// TIA Portal project "032_500_Analog_Values_V14" (V14)

(* hardware
DEVICE "S71500/ET200MP station_1"  S7-1500 station
   slot 0: "Rail_0"  Rack  6ES7 590-1***0-0AA0
   slot 0: "PM 190W 120/230VAC"  PM 190W 120/230VAC  6EP1333-4BA00
   slot 1: "CPU1516F"  CPU 1516F-3 PN/DP  6ES7 516-3FN01-0AB0  V2.1
      slot 3: "CPU display_1"  6ES7591-1BA00-0AA0
   slot 2: "DI 32x24VDC HF_1"  DI 32x24VDC HF  6ES7 521-1BL00-0AB0  V2.1
   slot 3: "DQ 32x24VDC/0.5A HF_1"  DQ 32x24VDC/0.5A HF  6ES7 522-1BL01-0AB0  V1.0
   slot 4: "AI 8xU/I/RTD/TC ST_1"  AI 8xU/I/RTD/TC ST  6ES7 531-7KF00-0AB0  V2.1
   slot 5: "AQ 4xU/I ST_1"  AQ 4xU/I ST  6ES7 532-5HD00-0AB0  V2.1
*)

// ===== PLC "CPU1516F"  CPU 1516F-3 PN/DP =====

VAR_GLOBAL   // PLC tag table "Tag table_sorting station"
   "-A1" AT %I0.0 : Bool;   // return signal emergency stop ok (nc)
   "-K0" AT %I0.1 : Bool;   // main switch „ON“ (no)
   "-S0" AT %I0.2 : Bool;   // mode selector manual(0) / automatic(1)
   "-S1" AT %I0.3 : Bool;   // pushbutton automatic start (no)
   "-S2" AT %I0.4 : Bool;   // pushbutton automatic stop (nc)
   "-B1" AT %I0.5 : Bool;   // sensor cylinder -M4 retracted (no)
   "-B2" AT %I0.6 : Bool;   // sensor cylinder -M4 extended (nc)
   "-B3" AT %I0.7 : Bool;   // sensor motor -M1 actice (pulse signal for positioning) (no)
   "-B4" AT %I1.0 : Bool;   // sensor part at slide (no)
   "-B5" AT %I1.1 : Bool;   // sensor metal part (no)
   "-B6" AT %I1.2 : Bool;   // sensor part in front of cylinder -M4 (no)
   "-B7" AT %I1.3 : Bool;   // sensor part at end of conveyor (no)
   "-S3" AT %I1.4 : Bool;   // pushbutton manual mode conveyor –M1 forwards (no)
   "-S4" AT %I1.5 : Bool;   // pushbutton manual mode conveyor –M1 backwards (no)
   "-S5" AT %I1.6 : Bool;   // pushbutton manual mode cylinder -M4 retract (no)
   "-S6" AT %I1.7 : Bool;   // pushbutton manual mode cylinder -M4 extend (no)
   "-Q1" AT %Q0.0 : Bool;   // conveyor motor -M1 forwards fixed speed
   "-Q2" AT %Q0.1 : Bool;   // conveyor motor -M1 backwards fixed speed
   "-Q3" AT %Q0.2 : Bool;   // conveyor motor -M1 variable speed
   "-M2" AT %Q0.3 : Bool;   // cylinder -M4 retract
   "-M3" AT %Q0.4 : Bool;   // cylinder -M4 extend
   "-P1" AT %Q0.5 : Bool;   // display „main switch on“
   "-P2" AT %Q0.6 : Bool;   // display „manual mode“
   "-P3" AT %Q0.7 : Bool;   // display „automatic mode“
   "-P4" AT %Q1.0 : Bool;   // display „emergency stop activated“
   "-P5" AT %Q1.1 : Bool;   // display „automatic mode started“
   "-P6" AT %Q1.2 : Bool;   // display cylinder -M4 „retracted“
   "-P7" AT %Q1.3 : Bool;   // display cylinder -M4 „extended“
   "-U1" AT %AW64 : Int;   // manipulated value speed in 2 directions +/- 10V / Stellwert Drehzahl des Motors in 2 Richtungen +/-10V entsprechen +/- 50 U/min
   "-B8" AT %EW64 : Int;   // sensor actual value speed 0 …10V / Sensor Istwert Drehzahl des Motors +/-10V entsprechen +/- 50 U/min
END_VAR

DATA_BLOCK "MOTOR_AUTO_DB"   // DB1
{ S7_Optimized_Access := 'TRUE' }
VERSION : 0.1
// stored: InstanceOfName MOTOR_AUTO
"MOTOR_AUTO"
BEGIN
END_DATA_BLOCK

FUNCTION_BLOCK "MOTOR_AUTO"   // FB1, FBD
TITLE = Motor control in automatic mode / Motoransteuerung im Automatikbetrieb
{ S7_Optimized_Access := 'TRUE' }
VERSION : 0.1
// Conveyor motor in automatic mode:
// The bit  Memory_automatic_start_stop is set with the input Start, but only if the reset conditions
// are not fufilled.
// The bit  Memory_automatic_start_stop is reset with the input Stop or if the safety shutoff is activated or if the automatic mode is not activated ( manual mode).
// If Memory_automatic_start_stop is set, the enable conditions are granted and Memory_conveyor_start_stop is set the output Conveyor_motor_automatic_mode is activated.
// For reasons of energy efficiency the conveyor motor should only run if a part is present.
// Therefore Memory_conveyor_start_stop is set if there is a part detected in front of Sensor_slide
// and reset with a negative edge at Sensor_end_of_conveyor or if the safety shutoff is activated
// or if the automatic mode is not activated ( manual mode).
// 
// As the Sensor_end_of_conveyor couldn't be assembled directly at the end of the conveyor we need
// an additional time until we can stop the motor.
// For that purpose we use an extended pulse timer in between the Sensor_end_of_conveyor
// and the negative edge detection.
// Bandmotor im Automatikbetrieb: 
// Der Speicher_Automatik_Start_Stopp wird mit dem Start_Befehl speichernd eingeschaltet, jedoch nur wenn die Rücksetzbedingungen nicht anstehen.  
// Der Speicher_Automatik_Start_Stopp wird wird zurückgesetzt, wenn der Stopp_Befehl ansteht oder die Schutzabschaltung aktiv ist oder der Automatikbetrieb nicht aktiviert ist (Handbetrieb).
// Der Ausgang Automatik_Motor wird angesteuert wenn der Speicher_Automatik_Start_Stopp gesetzt ist, die Freigabebedingungen erfüllt sind und der Speicher_Band_Start_Stopp gesetzt ist.
// Aus Energiespargründen soll das Band nur laufen wenn auch ein Teil vorhanden ist.
// Deshalb wird der Speicher_Band_Start_Stopp gesetzt wenn der Sensor_Rutsche_belegt ein Teil meldet und zurückgesetzt wenn der Sensor_Bandende eine negative Flanke erzeugt oder die Schutzabschaltung aktiv ist oder der Automatikbetrieb nicht aktiviert ist (Handbetrieb).
   VAR_INPUT
      Automatic_mode_active : Bool;   // Automatic mode activated / Betriebsart Automatikbetrieb aktiviert
      Start : Bool;   // Pushbutton automatic start / Start- Befehl für Automatikbetrieb
      Stop : Bool;   // Pushbutton automatic stop / Stopp- Befehl für Automatikbetrieb
      Enable_OK : Bool;   // All enable conditions OK / Alle Freigabebedingungen erfüllt
      Safety_shutoff_active : Bool;   // Safety shutoff active e.g. emergency stop operated / Schutzabschaltung aktiv z.B. Not Halt betätigt
      Sensor_slide : Bool;   // Sensor part at slide / Sensor Rutsche belegt
      Sensor_end_of_conveyor : Bool;   // Sensor part at end of conveyor / Sensor am Bandende
   END_VAR
   VAR_OUTPUT
      Conveyor_motor_automatic_mode : Bool;   // Control of the conveyor motor in automatic mode / Ansteuerung des Bandmotors im Automatikbetrieb
   END_VAR
   VAR
      Memory_automatic_start_stop : Bool;   // Memory used for start/ stop automatic mode / Speicher für Start- und Stoppfunktion im Automatikbetrieb
      Memory_conveyor_start_stop : Bool;   // Memory used for start/ stop of conveyor in automatic mode (energy saving) / Speicher für Start- und Stoppfunktion des Bandmotors(Energiesparmodus)
      Memory_edge_detection : Bool;   // Memory used for edge detection / Speicher für Flankenerkennung
      IEC_Timer_overrun : IEC_TIMER;
   END_VAR
   VAR RETAIN
      IEC_Counter_plastic : IEC_COUNTER;
   END_VAR
   VAR_TEMP   // added for the SCL form of the ladder/FBD networks
      _w1 : Bool;
   END_VAR
BEGIN

REGION Network 1: Overrun time end of conveyor pulse 2 seconds
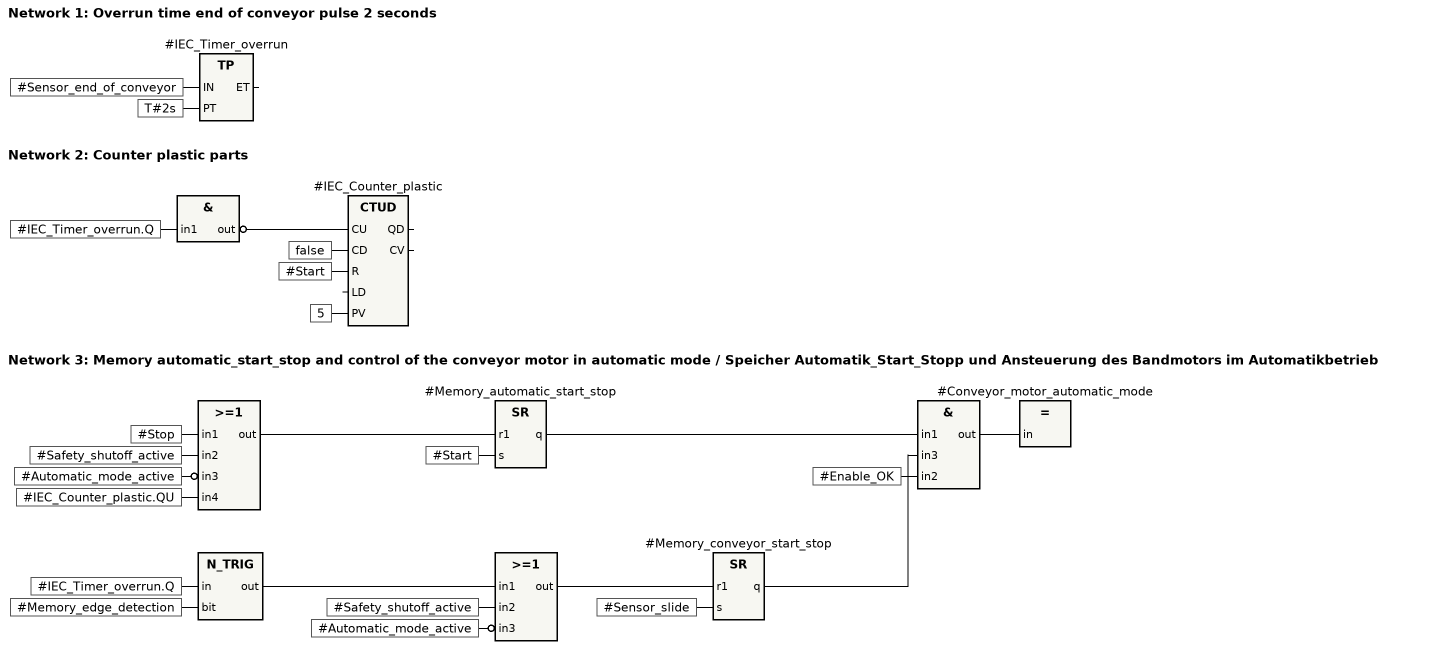
   #IEC_Timer_overrun.TP(IN := #Sensor_end_of_conveyor, PT := T#2s);
END_REGION

REGION Network 2: Counter plastic parts
   #IEC_Counter_plastic.CTUD(CU := NOT #IEC_Timer_overrun.Q, CD := false, R := #Start, PV := 5);
END_REGION

REGION Network 3: Memory automatic_start_stop and control of the conveyor motor in automatic mode / Speicher Automatik_Start_Stopp und Ansteuerung des Bandmotors im Automatikbetrieb
   IF #Start THEN
       #Memory_automatic_start_stop := TRUE;   // SR flip-flop
   END_IF;
   IF #Stop OR #Safety_shutoff_active OR NOT #Automatic_mode_active OR #IEC_Counter_plastic.QU THEN
       #Memory_automatic_start_stop := FALSE;
   END_IF;
   #_w1 := NOT #IEC_Timer_overrun.Q AND #Memory_edge_detection;   // falling edge
   #Memory_edge_detection := #IEC_Timer_overrun.Q;
   IF #Sensor_slide THEN
       #Memory_conveyor_start_stop := TRUE;   // SR flip-flop
   END_IF;
   IF #_w1 OR #Safety_shutoff_active OR NOT #Automatic_mode_active THEN
       #Memory_conveyor_start_stop := FALSE;
   END_IF;
   #Conveyor_motor_automatic_mode := #Memory_automatic_start_stop AND #Memory_conveyor_start_stop AND #Enable_OK;
END_REGION
END_FUNCTION_BLOCK

FUNCTION "MOTOR_SPEEDCONTROL" : Bool   // FC10, FBD
TITLE = Speed control via analog output / Drehzahlsteuerung über Analogausgang
{ S7_Optimized_Access := 'TRUE' }
VERSION : 0.1
   VAR_INPUT
      Setpoint_speed : Real;   // Drehzahlvorgabe in Umdrehungen pro Minute (Bereich: +/- 50 U/min)
   END_VAR
   VAR_OUTPUT
      Manipulated_variable_speed_AO : Int;   // Drehzahlstellwert zur Ausgabe an Analogausgang
   END_VAR
   VAR_TEMP
      Setpoint_speed_OK : Bool;   // Drehzahlsollwert im Bereich +/- 50 U/min
      Manipulated_variable_speed_Norm : Real;   // Drehzahlstellwert normiert 0...1
   END_VAR
   // Ret_Val : Return = FALSE wenn Drehzahlsollwert OK / Return = TRUE wenn Drehzahlsollwert nicht OK
BEGIN

REGION Network 1: check setpoint speed for correct input range +/- 50 r/min / Überprüfung des Drehzahlsollwertes auf korrekte Eingabe im Bereich +/- 50 U/min
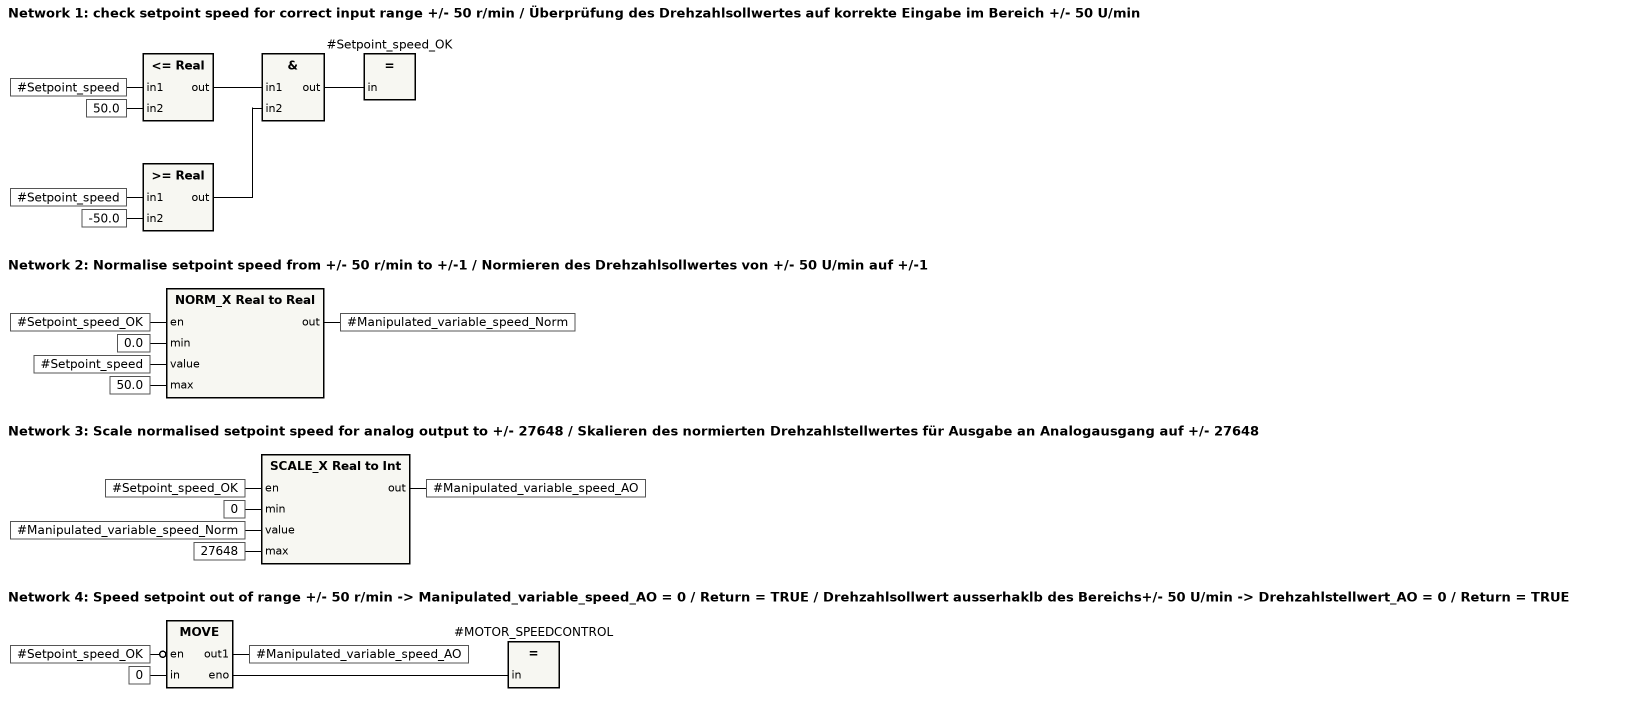
   #Setpoint_speed_OK := (#Setpoint_speed <= 50.0) AND (#Setpoint_speed >= (-50.0));
END_REGION

REGION Network 2: Normalise setpoint speed from +/- 50 r/min to +/-1 / Normieren des Drehzahlsollwertes von +/- 50 U/min auf +/-1
   IF #Setpoint_speed_OK THEN
       #Manipulated_variable_speed_Norm := NORM_X(MIN := 0.0, VALUE := #Setpoint_speed, MAX := 50.0);
   END_IF;
END_REGION

REGION Network 3: Scale normalised setpoint speed for analog output to +/- 27648 / Skalieren des normierten Drehzahlstellwertes für Ausgabe an Analogausgang auf +/- 27648
   IF #Setpoint_speed_OK THEN
       #Manipulated_variable_speed_AO := SCALE_X(MIN := 0, VALUE := #Manipulated_variable_speed_Norm, MAX := 27648);
   END_IF;
END_REGION

REGION Network 4: Speed setpoint out of range +/- 50 r/min -> Manipulated_variable_speed_AO = 0 / Return = TRUE / Drehzahlsollwert ausserhaklb des Bereichs+/- 50 U/min -> Drehzahlstellwert_AO = 0 / Return = TRUE
   IF NOT #Setpoint_speed_OK THEN #Manipulated_variable_speed_AO := 0; END_IF;
   #MOTOR_SPEEDCONTROL := NOT #Setpoint_speed_OK;
END_REGION
END_FUNCTION

FUNCTION "MOTOR_SPEEDMONITORING" : Void   // FC11, FBD
TITLE = Speed monitoring / Drehzahlüberwachung
{ S7_Optimized_Access := 'TRUE' }
VERSION : 0.1
   VAR_INPUT
      Actual_speed_AI : Int;   // Drehzahlistwert von Analogeingang
      Speed_limit_error_max : Real;   // Festlegung einer maximalen Drehzahl / Bei Überschreitung wird eine Störung ausgegeben
      Speed_limit_warning_max : Real;   // Festlegung einer maximalen Drehzahl / Bei Überschreitung wird eine Warnung ausgegeben
      Speed_limit_warning_min : Real;   // Festlegung einer minimalen Drehzahl / Bei Unterschreitung wird eine Warnung ausgegeben
      Speed_limit_error_min : Real;   // Festlegung einer minimalen Drehzahl / Bei Unterschreitung wird eine Störung ausgegeben
   END_VAR
   VAR_OUTPUT
      Error_max : Bool;   // Anzeige Störgrenze maximal wurde überschritten
      Warning_max : Bool;   // Anzeige Warngrenze maximal wurde überschritten
      Warning_min : Bool;   // Anzeige Warngrenze minimal wurde unterschritten
      Error_min : Bool;   // Anzeige Störgrenze minimal wurde unterschritten
      Actual_speed : Real;   // Drehzahlistwert skaliert zur Anzeige in Umdrehungen pro Minute (Bereich: +/- 50 U/min)
   END_VAR
   VAR_TEMP
      Actual_speed_norm : Real;   // Drehzahlistwert normiert 0...1
      Actual_speed_scaled : Real;   // Drehzahlistwert skaliert zur Verwendung im Baustein in Umdrehungen pro Minute (Bereich: +/- 50 U/min)
   END_VAR
BEGIN

REGION Network 1: Normalise actual speed from analog module to +/-1 / Normieren des Drehzahlistwertes von der Analogbaugruppe auf +/-1
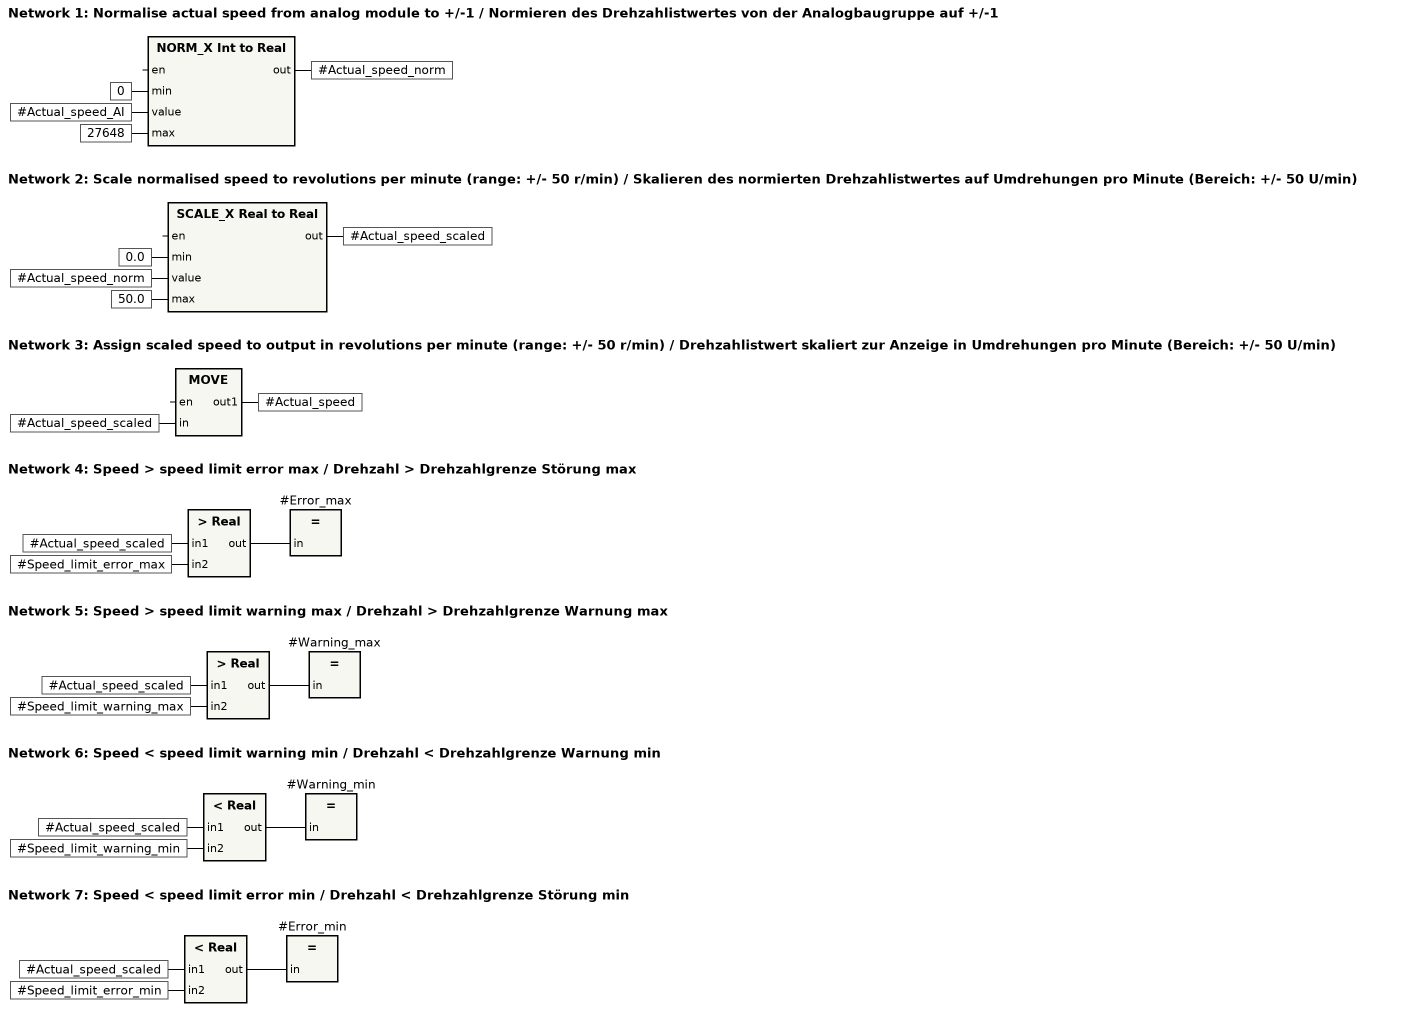
   #Actual_speed_norm := NORM_X(MIN := 0, VALUE := #Actual_speed_AI, MAX := 27648);
END_REGION

REGION Network 2: Scale normalised speed to revolutions per minute (range: +/- 50 r/min) / Skalieren des normierten Drehzahlistwertes auf Umdrehungen pro Minute (Bereich: +/- 50 U/min)
   #Actual_speed_scaled := SCALE_X(MIN := 0.0, VALUE := #Actual_speed_norm, MAX := 50.0);
END_REGION

REGION Network 3: Assign scaled speed to output in revolutions per minute (range: +/- 50 r/min) / Drehzahlistwert skaliert zur Anzeige in Umdrehungen pro Minute (Bereich: +/- 50 U/min)
   #Actual_speed := #Actual_speed_scaled;
END_REGION

REGION Network 4: Speed > speed limit error max / Drehzahl > Drehzahlgrenze Störung max
   #Error_max := #Actual_speed_scaled > #Speed_limit_error_max;
END_REGION

REGION Network 5: Speed > speed limit warning max / Drehzahl > Drehzahlgrenze Warnung max
   #Warning_max := #Actual_speed_scaled > #Speed_limit_warning_max;
END_REGION

REGION Network 6: Speed < speed limit warning min / Drehzahl < Drehzahlgrenze Warnung min
   #Warning_min := #Actual_speed_scaled < #Speed_limit_warning_min;
END_REGION

REGION Network 7: Speed < speed limit error min / Drehzahl < Drehzahlgrenze Störung min
   #Error_min := #Actual_speed_scaled < #Speed_limit_error_min;
END_REGION
END_FUNCTION

ORGANIZATION_BLOCK "Main"   // OB1, FBD, ProgramCycle
TITLE = "Main Program Sweep (Cycle)"
{ S7_Optimized_Access := 'TRUE' }
VERSION : 0.1
   VAR_INPUT
      Initial_Call : Bool;   // Initial call of this OB
      Remanence : Bool;   // =True, if remanent data are available
   END_VAR
   VAR_TEMP
      Motor_speed_monitoring_error_max : Bool;
      Motor_speed_monitoring_warning_max : Bool;
      Motor_speed_monitoring_warning_min : Bool;
      Motor_speed_monitoring_error_min : Bool;
      Motor_speed_monitoring_actual_speed : Real;
      Motor_speed_monitoring_Ret_Val : Bool;   // Rückgabewert (Return) des FCs MOTOR_DREHZAHLSTEUERUNG
   END_VAR
BEGIN

REGION Network 1: Speed monitoring conveyor motor / Drehzahlüberwachung Bandmotor
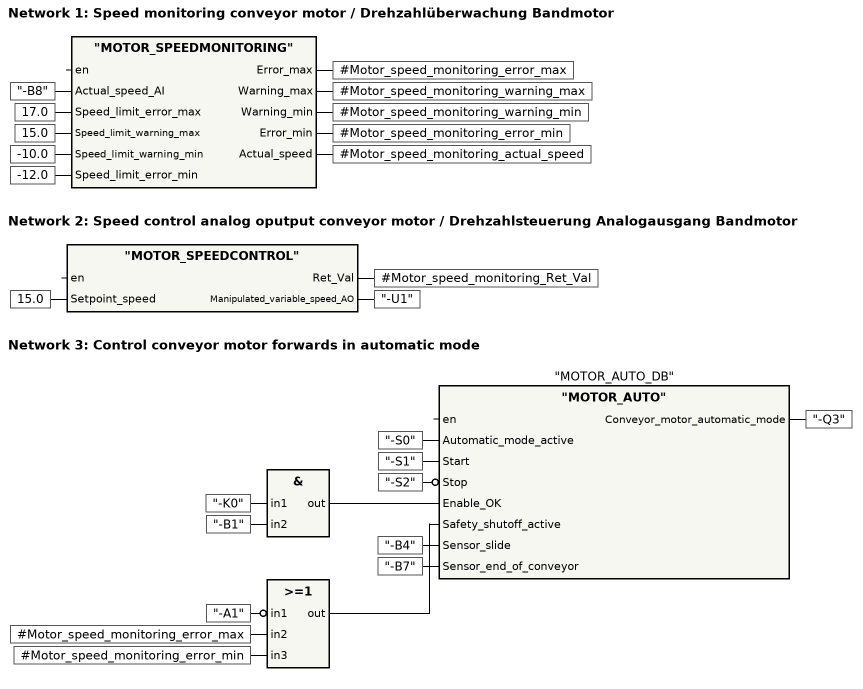
   "MOTOR_SPEEDMONITORING"(Actual_speed_AI := "-B8",
                           Speed_limit_error_max := 17.0,
                           Speed_limit_warning_max := 15.0,
                           Speed_limit_warning_min := -10.0,
                           Speed_limit_error_min := -12.0,
                           Error_max => #Motor_speed_monitoring_error_max,
                           Warning_max => #Motor_speed_monitoring_warning_max,
                           Warning_min => #Motor_speed_monitoring_warning_min,
                           Error_min => #Motor_speed_monitoring_error_min,
                           Actual_speed => #Motor_speed_monitoring_actual_speed);
END_REGION

REGION Network 2: Speed control analog oputput conveyor motor / Drehzahlsteuerung Analogausgang Bandmotor
   #Motor_speed_monitoring_Ret_Val := "MOTOR_SPEEDCONTROL"(Setpoint_speed := 15.0,
                           Manipulated_variable_speed_AO => "-U1");
END_REGION

REGION Network 3: Control conveyor motor forwards in automatic mode
   "MOTOR_AUTO_DB"(Automatic_mode_active := "-S0",   // "MOTOR_AUTO"
                   Start := "-S1",
                   Stop := NOT "-S2",
                   Enable_OK := "-K0" AND "-B1",
                   Safety_shutoff_active := NOT "-A1" OR #Motor_speed_monitoring_error_max OR #Motor_speed_monitoring_error_min,
                   Sensor_slide := "-B4",
                   Sensor_end_of_conveyor := "-B7",
                   Conveyor_motor_automatic_mode => "-Q3");
END_REGION
END_ORGANIZATION_BLOCK